FUNCTION Anolog_To_Height : real
VAR_INPUT
	value	:DINT;
END_VAR
VAR
	i	:INT;
	rel1,rel2	:REAL;
END_VAR

i:=0;

WHILE (HeightMap[i]<value AND HeightMap[i]>0) DO
	i:=i+1;
END_WHILE
i	:=LIMIT(1,i,380);
rel1:= TO_REAL(value-HeightMap[i-1]);
rel2:= rel1/LIMIT(1.0,TO_REAL(HeightMap[i]-HeightMap[i-1]),10000);

Anolog_To_Height:=LIMIT(0,TO_REAL(i-1)+rel2,380);

END_FUNCTION

(* stored: Version 1.1.0.1, ProductVersion 3.1.4024.12
   POU Anolog_To_Height: Id {e0caa4a9-4086-4aaf-bacd-ec7eb034e415}, SpecialFunc None *)
